FUNCTION_BLOCK F_N_MIN_MEAN_LREAL (* Stores arriving data and releases the mean in intervals specified by input N. *)
  (* Standard: 61499-2; Description: Stores arriving data and releases the mean in intervals specified by input N. The elapsed time between values is determined via the time stamp. Data should be sent at each interval N. Smaller intervals are also permitted. If the interval set by N is exceeded, a correction for the mean is corrected by factoring in the time N was exceeded by and the next computation is initialized with the data that was excluded. *)
  (* Version 1.0, 2017-06-13, Marc Jakobi, HTW Berlin *)
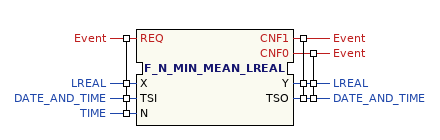
  EVENT_INPUT
    REQ WITH N, X, TSI; (* Normal Execution Request *)
  END_EVENT
  EVENT_OUTPUT
    CNF1 WITH Y, TSO; (* New average arrived *)
    CNF0 WITH Y, TSO; (* No new average arrived *)
  END_EVENT
  VAR_INPUT
    X : LREAL; (* Input data *)
    TSI : DATE_AND_TIME; (* Time stamp *)
    N : TIME; (* Time interval of mean *)
  END_VAR
  VAR_OUTPUT
    Y : LREAL; (* N minute mean of X *)
    TSO : DATE_AND_TIME; (* Time stamp *)
  END_VAR
  FBS
    F_SUB_DT_DT : F_SUB_DT_DT;
    LAST_TS : FB_SHIFT1_DT;
    RESET_CHK : F_LT;
    EO0_RESET : E_SWITCH;
    E_SPLIT : E_SPLIT;
    E_SPLIT_1 : E_SPLIT;
    E_REND : E_REND;
    TIME_FACTOR : F_DIV;
    F_MUL : F_MUL;
    LREAL2LREAL_1 : LREAL2LREAL;
    F_TIME_TO_ULINT_1 : F_TIME_TO_LREAL;
    F_TIME_TO_ULINT : F_TIME_TO_LREAL;
    LREAL2LREAL_2 : LREAL2LREAL;
    LREAL2LREAL_3 : LREAL2LREAL;
    E_SWITCH : E_SWITCH;
    SUB : F_SUB_DT_DT;
    F_TIME_TO_LREAL : F_TIME_TO_LREAL;
    F_GT : F_GT(IN2 := LREAL#0);
    ACCUMULATE_DATA : F_ACCUM_LREAL(INIT := LREAL#0);
    E_REND_1 : E_REND;
    E_SPLIT_2 : E_SPLIT;
    OVERTIME : F_SUB;
    OVERTIME_FACTOR : F_DIV;
    TIME2LREAL : F_TIME_TO_LREAL;
    LREAL2LREAL : LREAL2LREAL;
    OVERTIME_DATA : F_SUB;
    ACCUMULATE_TIME : F_ACCUM_TIME(INIT := T#0ms);
    RESET : E_SPLIT_3;
    INIT_TO_OVERTIME : TIME2TIME;
    ONE__PLUS_OVERTIME_FACTOR : F_ADD(IN2 := LREAL#1);
    LREAL2LREAL_4 : LREAL2LREAL;
    LREAL2LREAL_5 : LREAL2LREAL;
    N_MIN_MEAN : F_DIV;
    F_SUB_DT_TIME : F_SUB_DT_TIME;
    INITIALIZE : E_SPLIT;
    E_MERGE : E_MERGE;
    E_INIT_CHK : E_INIT_CHK;
    LIMIT_OVERTIME : F_MIN;
    RESET_DATA_IF_TOO_MUCH_OVERTIME : F_GT;
    RESET_DATA_IF_TOO_MUCH_OVERTIME2 : F_SEL(IN1 := LREAL#0);
    LREAL2LREAL_6 : LREAL2LREAL;
  END_FBS
  EVENT_CONNECTIONS
    RESET_CHK.CNF TO EO0_RESET.EI;
    REQ TO E_SPLIT.EI;
    E_SPLIT.EO1 TO LAST_TS.REQ;
    F_SUB_DT_DT.CNF TO E_SPLIT_1.EI;
    E_REND.EO TO TIME_FACTOR.REQ;
    E_SPLIT.EO2 TO F_TIME_TO_ULINT_1.REQ;
    F_TIME_TO_ULINT_1.CNF TO E_REND.EI2;
    E_SPLIT_1.EO2 TO F_TIME_TO_ULINT.REQ;
    F_TIME_TO_ULINT.CNF TO E_REND.EI1;
    F_MUL.CNF TO LREAL2LREAL_1.REQ;
    TIME_FACTOR.CNF TO LREAL2LREAL_2.REQ;
    LREAL2LREAL_2.CNF TO F_MUL.REQ;
    SUB.CNF TO F_TIME_TO_LREAL.REQ;
    F_TIME_TO_LREAL.CNF TO F_GT.REQ;
    F_GT.CNF TO E_SWITCH.EI;
    E_SWITCH.EO1 TO F_SUB_DT_DT.REQ;
    LREAL2LREAL_1.CNF TO ACCUMULATE_DATA.REQ;
    ACCUMULATE_DATA.CNF TO E_REND_1.EI2;
    E_REND_1.EO TO RESET_CHK.REQ;
    E_SPLIT_2.EO2 TO E_REND.R;
    E_SWITCH.EO0 TO E_SPLIT_2.EI;
    E_SPLIT_2.EO1 TO E_REND_1.R;
    EO0_RESET.EO0 TO OVERTIME.REQ;
    TIME2LREAL.CNF TO OVERTIME_FACTOR.REQ;
    OVERTIME_FACTOR.CNF TO LREAL2LREAL.REQ;
    LREAL2LREAL_3.CNF TO OVERTIME_DATA.REQ;
    E_SPLIT_1.EO1 TO ACCUMULATE_TIME.REQ;
    ACCUMULATE_TIME.CNF TO E_REND_1.EI1;
    OVERTIME.CNF TO INIT_TO_OVERTIME.REQ;
    LREAL2LREAL.CNF TO ONE__PLUS_OVERTIME_FACTOR.REQ;
    ONE__PLUS_OVERTIME_FACTOR.CNF TO LREAL2LREAL_4.REQ;
    LREAL2LREAL_5.CNF TO RESET.EI;
    LREAL2LREAL_4.CNF TO N_MIN_MEAN.REQ;
    N_MIN_MEAN.CNF TO LREAL2LREAL_3.REQ;
    INIT_TO_OVERTIME.CNF TO F_SUB_DT_TIME.REQ;
    F_SUB_DT_TIME.CNF TO TIME2LREAL.REQ;
    RESET.E1 TO E_MERGE.EI2;
    INITIALIZE.EO1 TO LAST_TS.REQ;
    INITIALIZE.EO2 TO E_MERGE.EI1;
    E_MERGE.EO TO CNF1;
    EO0_RESET.EO1 TO CNF0;
    LAST_TS.CNF TO E_INIT_CHK.REQ;
    E_INIT_CHK.INIT TO INITIALIZE.EI;
    E_INIT_CHK.NOINIT TO SUB.REQ;
    RESET.E3 TO LIMIT_OVERTIME.REQ;
    LIMIT_OVERTIME.CNF TO RESET_DATA_IF_TOO_MUCH_OVERTIME.REQ;
    OVERTIME_DATA.CNF TO LREAL2LREAL_6.REQ;
    LREAL2LREAL_6.CNF TO LREAL2LREAL_5.REQ;
    RESET_DATA_IF_TOO_MUCH_OVERTIME.CNF TO ACCUMULATE_TIME.R;
    RESET.E2 TO RESET_DATA_IF_TOO_MUCH_OVERTIME2.REQ;
    RESET_DATA_IF_TOO_MUCH_OVERTIME2.CNF TO ACCUMULATE_DATA.R;
  END_CONNECTIONS
  DATA_CONNECTIONS
    TSI TO LAST_TS.I;
    LAST_TS.O1 TO F_SUB_DT_DT.IN1;
    LAST_TS.O2 TO F_SUB_DT_DT.IN2;
    N TO RESET_CHK.IN2;
    RESET_CHK.OUT TO EO0_RESET.G;
    N TO F_TIME_TO_ULINT_1.IN;
    F_TIME_TO_ULINT_1.OUT TO TIME_FACTOR.IN2;
    F_SUB_DT_DT.OUT TO F_TIME_TO_ULINT.IN;
    F_TIME_TO_ULINT.OUT TO TIME_FACTOR.IN1;
    F_MUL.OUT TO LREAL2LREAL_1.IN;
    TIME_FACTOR.OUT TO LREAL2LREAL_2.IN;
    LAST_TS.O1 TO SUB.IN1;
    LAST_TS.O2 TO SUB.IN2;
    SUB.OUT TO F_TIME_TO_LREAL.IN;
    F_TIME_TO_LREAL.OUT TO F_GT.IN1;
    F_GT.OUT TO E_SWITCH.G;
    LREAL2LREAL_1.OUT TO ACCUMULATE_DATA.IN;
    N TO OVERTIME.IN2;
    OVERTIME.OUT TO TIME2LREAL.IN;
    TIME2LREAL.OUT TO OVERTIME_FACTOR.IN1;
    F_TIME_TO_ULINT_1.OUT TO OVERTIME_FACTOR.IN2;
    X TO F_MUL.IN2;
    LREAL2LREAL_2.OUT TO F_MUL.IN1;
    OVERTIME_FACTOR.OUT TO LREAL2LREAL.IN;
    F_SUB_DT_DT.OUT TO ACCUMULATE_TIME.IN;
    ACCUMULATE_TIME.OUT TO RESET_CHK.IN1;
    ACCUMULATE_TIME.OUT TO OVERTIME.IN1;
    OVERTIME.OUT TO INIT_TO_OVERTIME.IN;
    ACCUMULATE_DATA.OUT TO OVERTIME_DATA.IN1;
    LREAL2LREAL_3.OUT TO OVERTIME_DATA.IN2;
    LREAL2LREAL.OUT TO ONE__PLUS_OVERTIME_FACTOR.IN1;
    ONE__PLUS_OVERTIME_FACTOR.OUT TO LREAL2LREAL_4.IN;
    LREAL2LREAL_5.OUT TO Y;
    N_MIN_MEAN.OUT TO LREAL2LREAL_3.IN;
    ACCUMULATE_DATA.OUT TO N_MIN_MEAN.IN1;
    LREAL2LREAL_4.OUT TO N_MIN_MEAN.IN2;
    LREAL2LREAL_3.OUT TO LREAL2LREAL_5.IN;
    TSI TO F_SUB_DT_TIME.IN1;
    INIT_TO_OVERTIME.OUT TO F_SUB_DT_TIME.IN2;
    F_SUB_DT_TIME.OUT TO TSO;
    N TO LIMIT_OVERTIME.IN2;
    INIT_TO_OVERTIME.OUT TO LIMIT_OVERTIME.IN1;
    LIMIT_OVERTIME.OUT TO ACCUMULATE_TIME.INIT;
    INIT_TO_OVERTIME.OUT TO RESET_DATA_IF_TOO_MUCH_OVERTIME.IN1;
    N TO RESET_DATA_IF_TOO_MUCH_OVERTIME.IN2;
    RESET_DATA_IF_TOO_MUCH_OVERTIME.OUT TO RESET_DATA_IF_TOO_MUCH_OVERTIME2.G;
    OVERTIME_DATA.OUT TO LREAL2LREAL_6.IN;
    LREAL2LREAL_6.OUT TO RESET_DATA_IF_TOO_MUCH_OVERTIME2.IN0;
    RESET_DATA_IF_TOO_MUCH_OVERTIME2.OUT TO ACCUMULATE_DATA.INIT;
  END_CONNECTIONS
END_FUNCTION_BLOCK
